ABB RobotStudio station: Welding_robots.rsstnx

Station Welding_robots (saved by RobotStudio 23.4.10609.1)
Controller IRB1600_Controler_1, task T_ROB1: task frame (RAPID world) sits at (2310, 0, 450) mm, rotated rx 0 ry 0 rz 180 deg in the station
Controller IRB1600_Controler_0, task T_ROB1: task frame (RAPID world) sits at (-100, 0, 250) mm in the station
Controller IRB1600_Controler_0
  mechanical unit ROB_1: IRB1600_0, 6 joints, base frame (0, 0, 0) mm
Controller IRB1600_Controler_1
  mechanical unit ROB_1: IRB1600_1, 6 joints, base frame (0, 0, 0) mm
Layout (positions relative to the parent item):
  - IRB1600_0 [mechanism, from %ABB.RobotStudio.Models.IRB1600%\IRB1600_6_120_G_02.rslib] at (-100, 0, 250) mm; joint values [0.6531, 0.5914, 0.0625, -1.1196, 1.1483, 3.1244] (rad or m)
  - IRB1600_1 [mechanism, from %ABB.RobotStudio.Models.IRB1600%\IRB1600_6_120_G_02.rslib] at (2310, 0, 450) mm, rotated rx 0 ry 0 rz 180 deg; joint values [0, 0, 0, 0, 0.5236, 0] (rad or m)
  - Welding_tool_0 [mechanism, from %ABB.RobotStudio.Models.ArcWelding%\Fronius_Robacta_MTG4000_22deg.rslib] at (644.43, 502.38, 729.15) mm, rotated rx 128.63 ry 25.15 rz 61.99 deg
  - Welding_tool_1 [mechanism, from %ABB.RobotStudio.Models.ArcWelding%\Fronius_Robacta_MTG4000_22deg.rslib] at (1503.71, 0, 1379) mm, rotated rx 180 ry 60 rz 0 deg
  - Conveyor [part, from %ABB.RobotStudio.Models.Conveyors%\Conveyor 950 4000 h2.rslib] at (1650, -2000, 0) mm, rotated rx 0 ry 0 rz 90 deg
  - Placa_0 [graphiccomponentgroup] at (800, -600, 430) mm
    - Pieza_3 [part] at (200, 200, 50) mm, size 300 x 298.4 x 100 mm
    - Pieza_2 [part] at (550, 50, 50) mm, rotated rx 0 ry 0 rz 70 deg, size 500 x 100 x 50 mm
    - Pieza_4 [part] at (200, 400, 85) mm, rotated rx -45 ry 0 rz 90 deg, size 500 x 100 x 50 mm
    - Pieza_5 [part] at (500, 750, 50) mm, size 400 x 397.8 x 100 mm
    - Pieza_1 [part] at (-800, 600, -400) mm, size 800 x 1200 x 50 mm
  - IRB1600_base_0 [part] at (-500, -450, -200) mm, size 700 x 700 x 450 mm
  - IRB1600_base_1 [part] at (2050, -450, 0) mm, size 700 x 700 x 450 mm
  - Grupo_1 [graphiccomponentgroup]
  - Sistema de coordenadas_4 [frame] at (800, -600, 479.99) mm
Attachment: Welding_tool_1 is attached to IRB1600_1 / Link6
Attachment: Welding_tool_0 is attached to IRB1600_0 / Link6
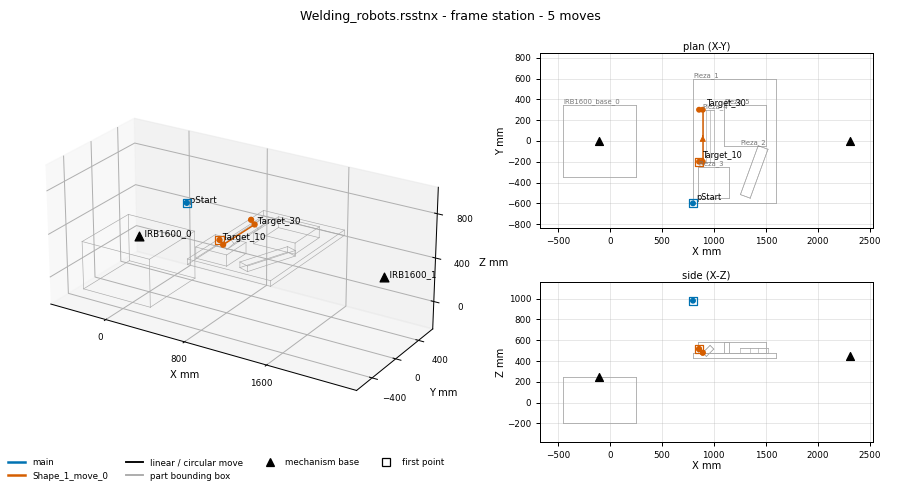
[picture p0: tool path of Welding_robots.rsstnx in frame station, 5 of 5 moves have a stored position in this frame; points joined in program order, loops and branches not executed]
Targets, tools, work objects and paths stored in the station, written as RAPID:
! task T_ROB1
MODULE MainModule
  CONST robtarget pHome:=[[200,0,200],[0,0,1,0],[0,0,0,0],[9E+09,9E+09,9E+09,9E+09,9E+09,9E+09]];
  CONST jointtarget jtHome:=[[0,0,0,0,0,0],[9E+09,9E+09,9E+09,9E+09,9E+09,9E+09]];
  CONST robtarget pStart:=[[0,0,500],[0,0,1,0],[0,0,0,0],[9E+09,9E+09,9E+09,9E+09,9E+09,9E+09]];
  CONST robtarget pStart_1:=[[0,400,500],[0,0,1,0],[0,0,0,0],[9E+09,9E+09,9E+09,9E+09,9E+09,9E+09]];
  PROC main()
    MoveJ pStart,v1000,fine,Weldgun\WObj:=Level_0;
    Shape_1_Move_0;
  ENDPROC
ENDMODULE

! task T_ROB1
MODULE CalibData
  PERS tooldata Weldgun:=[TRUE,[[20.31,0,363.689],[0.948464781,0,0.316882565,0]],[1,[0,0,1],[1,0,0,0],0,0,0]];
  TASK PERS wobjdata Level_0:=[FALSE,TRUE,"",[[900,-599.9,229.854],[1,0,0,0]],[[0,0,0],[1,0,0,0]]];
  TASK PERS wobjdata Tilt_45:=[FALSE,TRUE,"",[[994.289,-200,230],[0.923879533,0,0.382683432,0]],[[0,0,0],[1,0,0,0]]];
ENDMODULE

! task T_ROB1
MODULE Shape_0
  PROC Shape_0_move_0()
  ENDPROC
ENDMODULE

! task T_ROB1
MODULE Shape_1
  CONST robtarget Target_10:=[[-49.999772396,0,-0.50229766],[0.38,0.38,0.596,0.596],[0,0,0,0],[9E+09,9E+09,9E+09,9E+09,9E+09,9E+09]];
  CONST robtarget Target_20:=[[0.000227604,0,-0.502297712],[0.38,0.38,0.596,0.596],[0,0,0,0],[9E+09,9E+09,9E+09,9E+09,9E+09,9E+09]];
  CONST robtarget Target_30:=[[0.000227604,500,-0.502297712],[0.38,0.38,0.596,0.596],[0,0,0,0],[9E+09,9E+09,9E+09,9E+09,9E+09,9E+09]];
  CONST robtarget Target_40:=[[-49.999772396,500,-0.50229766],[0.5,0.5,0.5,0.5],[0,0,0,0],[9E+09,9E+09,9E+09,9E+09,9E+09,9E+09]];
  PROC Shape_1_move_0()
    MoveL Target_10,v1000,fine,Weldgun\WObj:=Tilt_45;
    MoveL Target_20,v1000,fine,Weldgun\WObj:=Tilt_45;
    MoveL Target_30,v1000,fine,Weldgun\WObj:=Tilt_45;
    MoveL Target_40,v1000,z100,Weldgun\WObj:=Tilt_45;
  ENDPROC
ENDMODULE

! task T_ROB1
MODULE CalibData
  PERS tooldata Weldgun:=[TRUE,[[20.31,0,363.689],[0.948464781,0,0.316882565,0]],[1,[0,0,1],[1,0,0,0],0,0,0]];
ENDMODULE

! task T_ROB1
MODULE Module1
  PROC main()
  ENDPROC
ENDMODULE

